FUNCTION F_KontrollZeiten : BOOL
VAR_INPUT
END_VAR
VAR
	bTmp : BOOL;
	localWord:WORD;
END_VAR

(* Netzwerk: 1 *** Kontroll-Zeiten *)

//ToDo: den Sinn der Aktion herausbekommen...
//evtl. Bitmuster auf dem AW erkennen...
(*
L AW 0 -- Akku 1 nach Akku 2, dann AW0 in Akku 1 -- AW0 offensichtlich Ausgangswort 0
T LW 0 -- Akku 1 nach LW 0 -- Ausgangswort0 in LW 0 speichern
L "DB6".d408 DB6.DBD408 -- Zuw.v. AW0 -- Akku 1 nach Akku 2, dann "DB6".d408 in Akku 1

L LD 0 -- Akku 1 nach Akku 2, dann LD 0 in Akku 1 -- Frage, was steht in LD 0 (Lokaldaten-Doppelwort (LD))

T "DB6".d408 DB6.DBD408 -- Zuw.v. AW0 -- T beeinflusst nichts...

-- [XOD] ... Bei der Verknüpfung von Doppelwörtern wird der Inhalt von AKKU 2 mit dem Inhalt von AKKU 1 verknüpft.
--  Das Verknüpfungsergebnis wird in AKKU 1 gespeichert, wobei der alte Inhalt überschrieben wird.

XOD

L 2# 11000000 11111111 00000000 00000000 -- Akku 1 nach Akku 2, dann Zahl in Akku 1
UD -- UND-Doppelwort
L 0
==D
*)

//Versuch...die Maske L 2# 110... kann wahrscheinlich entfallen, da ich das beim Füllen von IO.outWord0 schon
//berücksichtige NBT 2021-01-28

bTmp := (DB6.outWordAlt XOR IO.outWord0) <> 0; //ToDo: ergebnis dieser Aktion

(*
L S5T#1S200MS
SE "T 3" T3 -- Fehler-Kontr.Maschine (keine Bewegung) -- Zeit mit Einschaltverzögerung starten
L S5T#1S600MS
SE "T 15" T15 -- Verz. Endschalter-Brückung StSt *)

GVL.tonFehlerKontrMaschine( IN := bTmp, PT := T#1S200MS);

GVL.tonEndschalterBrueck( IN := bTmp, PT := T#1S600MS);

DB6.outWordAlt := IO.outWord0;

END_FUNCTION

(* stored: Version 1.1.0.1, ProductVersion 3.1.4024.3
   POU F_KontrollZeiten: Id {e0e17fcb-4403-4087-a554-9696ff5c6855}, SpecialFunc None *)
